FUNCTION_BLOCK FB_Camera EXTENDS FB_GCodeTool
VAR_INPUT
END_VAR
VAR_OUTPUT
END_VAR
VAR
	//SpecProperties
	rWorkingDistance		: REAL;
	bInvertWorkingDistance 	: BOOL;
	eLightOutput 			: E_TriggerOutput;
	nLightOutputChannel		: USINT;
	
	bCameraLightOn			: BOOL;
	
	bTakePicture			: BOOL;
	nStateA_TakePicture		: USINT;
	tDelayTakePicture		: TIME;
	timerTakePicture		: TON;
	nRequestArg1			: DINT;
	nRequestArg2			: DINT;
	nRequestArg3			: DINT;
	nRequestArg4			: DINT;	
END_VAR

IF bCameraLightOn THEN
	IF eLightOutput = E_TriggerOutput.MultiZOutput THEN
		fbMultiZDigiOut.M_On(nLightOutputChannel);
	ELSIF eLightOutput = E_TriggerOutput.MultiZPWM THEN
		fbMultiZPWM.M_On(nLightOutputChannel, 1000);
	END_IF
END_IF

IF eCurrentState = E_MachineState.MACHINESTATE_Active THEN
	IF bTakePicture THEN
		A_TakePicture();
		IF nStateA_TakePicture = 80 THEN
			nStateA_TakePicture := 0;
			bTakePicture := FALSE;
			M_RemoveListEntry(nSearchValue:= E_Action.ACTION_TakePicture);
		END_IF
	END_IF	
END_IF

SUPER^();

stProcessData.n32Data[7] := BOOL_TO_DINT(bCameraLightOn);
aObjProcData[nNotifyId] := stProcessData;

ACTION A_Reset:
nStateA_ResetSpec := 80;
SUPER^.A_Reset();
END_ACTION

ACTION A_Stop:
IF nStateA_Stop = 0 THEN
	IF bTakePicture AND nStateA_TakePicture < 70 THEN
		nStateA_TakePicture := 70;
	END_IF
	nStateA_Stop := 1;
END_IF

SUPER^.A_Stop();
END_ACTION

ACTION A_TakePicture:
IF nStateA_TakePicture = 0 THEN //Timer starten
	timerTakePicture(IN:= TRUE, PT:= tDelayTakePicture);
	IF timerTakePicture.Q THEN
		timerTakePicture(IN:= FALSE);
		stInterResponse.eInteractMessageType := E_InteractMessageType.INTERACTMES_NONE;
		stInteractRequest.eInteractMessageType := E_InteractMessageType.INTERACTMES_WaitForUser;
		stInteractRequest.nObjectId := nObjectID;
		stInteractRequest.nArg1 := nRequestArg1;
		stInteractRequest.nArg2 := nRequestArg2;
		stInteractRequest.nArg3 := nRequestArg3;
		stInteractRequest.nArg4 := nRequestArg4;
		nStateA_TakePicture := 1;
	END_IF
ELSIF nStateA_TakePicture = 1 THEN //Auf InteractResponse warten
	IF stInterResponse.eInteractMessageType = E_InteractMessageType.INTERACTMES_Continue OR 
							stInterResponse.eInteractMessageType = E_InteractMessageType.INTERACTMES_Cancel THEN
		stInteractRequest.eInteractMessageType := E_InteractMessageType.INTERACTMES_NONE;
		nStateA_TakePicture := 80;
	END_IF
ELSIF nStateA_TakePicture = 70 THEN //Abbrechen
	timerTakePicture(IN:= FALSE);
	stInteractRequest.eInteractMessageType := E_InteractMessageType.INTERACTMES_NONE;
	nStateA_TakePicture := 80;
END_IF
END_ACTION

METHOD FB_init : BOOL
VAR_INPUT
	bInitRetains : BOOL; // if TRUE, the retain variables are initialized (warm start / cold start)
	bInCopyCode : BOOL;  // if TRUE, the instance afterwards gets moved into the copy code (online change)
END_VAR
eObjectType := E_ObjectType.OBJECTTYPE_Camera;
eObjectGroup := E_ObjectGroup.OBJECTGROUP_MzTool OR E_ObjectGroup.OBJECTGROUP_Device;
END_METHOD

METHOD M_AddChild : ERRORID
VAR_INPUT
	pObject : POINTER TO FB_Object;
	nSlotNr	: UINT;	
	nIndex : INT;
END_VAR
//Kann folgende Objekte aufnehmen:
//Camera, Exposure
IF pObject > 0 THEN
	IF pObject^.P_eObjectType = E_ObjectType.OBJECTTYPE_Camera OR
		pObject^.P_eObjectType = E_ObjectType.OBJECTTYPE_DummyTool OR
		pObject^.P_eObjectType = E_ObjectType.OBJECTTYPE_Exposure THEN
		M_AddChild := SUPER^.M_AddChild(pObject,nSlotNr,nIndex);
	ELSE
		M_AddChild := E_ErrorIdObjMgmt.ERRORID_InvalidParentObject;
	END_IF
ELSE
	M_AddChild := E_ErrorIdObjMgmt.ERRORID_InvalidParentObject;
END_IF
END_METHOD

METHOD M_CancelAction
VAR_INPUT
	eAction : E_Action;
END_VAR
IF eAction = E_Action.ACTION_TakePicture THEN
	IF bTakePicture AND nStateA_TakePicture < 70 THEN
		nStateA_TakePicture := 70;
	END_IF
ELSE
	SUPER^.M_CancelAction(eAction);
END_IF
END_METHOD

METHOD M_CheckAction : ERRORID
VAR_INPUT
	refActionData 	: REFERENCE TO ST_ActionData;
	pCorrelObject	: POINTER TO FB_Object;
END_VAR

VAR
	pTarget : POINTER TO FB_TargetBase;
	pRack	: POINTER TO FB_Rack;
	pSlot	: POINTER TO FB_PieceSlot;
END_VAR
IF refActionData.eAction = E_Action.ACTION_TakePicture THEN
	RETURN;
ELSE
	M_CheckAction := SUPER^.M_CheckAction(refActionData, pCorrelObject);
END_IF
END_METHOD

METHOD M_ExeAction : ERRORID
VAR_INPUT
	refActionData : REFERENCE TO ST_ActionData;	
END_VAR
IF NOT (eCurrentState = E_MachineState.MACHINESTATE_Idle OR
	eCurrentState = E_MachineState.MACHINESTATE_Active OR
	eCurrentState = E_MachineState.MACHINESTATE_Ready) THEN
	M_ExeAction := E_ErrorIdCmd.ERRORID_InvalidState;
	RETURN;
END_IF

IF refActionData.eAction = E_Action.ACTION_SwitchLight THEN
	bCameraLightOn := DINT_TO_BOOL(refActionData.aParams[1]);
ELSIF refActionData.eAction = E_Action.ACTION_TakePicture THEN
	IF NOT bTakePicture THEN
		tDelayTakePicture := DINT_TO_TIME(refActionData.aParams[1]);
		nRequestArg1 := refActionData.aParams[2];
		nRequestArg2 := refActionData.aParams[3];
		nRequestArg3 := refActionData.aParams[4];
		nRequestArg4 := refActionData.aParams[5];
		
		fbList.A_AddHeadValue(hList := hList, putValue := E_Action.ACTION_TakePicture);
		bTakePicture := TRUE;
	END_IF
ELSE
	M_ExeAction := SUPER^.M_ExeAction(refActionData);
	RETURN;	
END_IF

bBusy := TRUE;
eCurrentState := E_MachineState.MACHINESTATE_Active;
END_METHOD

METHOD M_GetAllProps : ERRORID
VAR_INPUT
	refCmdData : REFERENCE TO  ST_CmdData;
END_VAR
SUPER^.M_GetAllProps(refCmdData);
nCurrentPropIndex := nCurrentPropIndex + 1;
refCmdData.n32Data[nCurrentPropIndex] := REAL_TO_DINT(rWorkingDistance);
nCurrentPropIndex := nCurrentPropIndex + 1;
refCmdData.n32Data[nCurrentPropIndex] := BOOL_TO_DINT(bInvertWorkingDistance);
nCurrentPropIndex := nCurrentPropIndex + 1;
refCmdData.n32Data[nCurrentPropIndex] := eLightOutput;
nCurrentPropIndex := nCurrentPropIndex + 1;
refCmdData.n32Data[nCurrentPropIndex] := nLightOutputChannel;
END_METHOD

METHOD M_SetAllProps : ERRORID
VAR_INPUT
	refCmdData : REFERENCE TO  ST_CmdData;
END_VAR
M_SetAllProps := SUPER^.M_SetAllProps(refCmdData);

IF M_SetAllProps > 0 THEN
	RETURN;
END_IF

//WorkingDistance
nCurrentPropIndex := nCurrentPropIndex + 1;
nSpecPropIndex := nCurrentPropIndex;
rWorkingDistance := DINT_TO_REAL(refCmdData.n32Data[nCurrentPropIndex]);
nCurrentPropIndex := nCurrentPropIndex + 1;
bInvertWorkingDistance := DINT_TO_BOOL(refCmdData.n32Data[nCurrentPropIndex]);

//LightOutput
nCurrentPropIndex := nCurrentPropIndex + 1;
eLightOutput := DINT_TO_USINT(refCmdData.n32Data[nCurrentPropIndex]);

//LightOutputChannel
nCurrentPropIndex := nCurrentPropIndex + 1;
nLightOutputChannel := DINT_TO_USINT(refCmdData.n32Data[nCurrentPropIndex]);

nNoOfProps := nCurrentPropIndex + 1;
END_METHOD

METHOD M_SetSingleProp : ERRORID
VAR_INPUT
	refCmdData : REFERENCE TO  ST_CmdData;
END_VAR
IF nSpecPropIndex = refCmdData.aHeader[1] THEN
	rWorkingDistance := DINT_TO_REAL(refCmdData.n32Data[0]);
ELSIF nSpecPropIndex + 1 = refCmdData.aHeader[1] THEN
	bInvertWorkingDistance := DINT_TO_BOOL(refCmdData.n32Data[0]);
ELSIF nSpecPropIndex + 3 = refCmdData.aHeader[1] THEN
	nLightOutputChannel := DINT_TO_USINT(refCmdData.n32Data[0]);
ELSE
	M_SetSingleProp := SUPER^.M_SetSingleProp(refCmdData);
END_IF
END_METHOD

PROPERTY P_stAbsPosTotal : ST_3DPoint
GET
VAR
	stPosTemp : ST_3DPoint;
END_VAR
stPosTemp := SUPER^.P_stAbsPosPhys;
IF bInvertWorkingDistance THEN
	stPosTemp.Z := stPosTemp.Z + rWorkingDistance;
ELSE
	stPosTemp.Z := stPosTemp.Z - rWorkingDistance;
END_IF
P_stAbsPosTotal := stPosTemp;
END_GET
END_PROPERTY

PROPERTY P_stCurrentPosTotal : ST_3DPoint
GET
VAR
	stPosTemp : ST_3DPoint;
END_VAR
stPosTemp := P_stCurrentPosPhys;
IF bInvertWorkingDistance THEN
	stPosTemp.Z := stPosTemp.Z + rWorkingDistance;
ELSE
	stPosTemp.Z := stPosTemp.Z - rWorkingDistance;
END_IF
P_stCurrentPosTotal := stPosTemp;
END_GET
END_PROPERTY

END_FUNCTION_BLOCK

(* stored: Version 1.1.0.1, ProductVersion 3.1.4024.11
   POU FB_Camera: Id {6d1727e9-21d6-47ab-aac6-925ca4a23f77}, SpecialFunc None
   Action A_Reset: Id {43cf20d4-7297-4beb-a482-862479609b93}
   Action A_Stop: Id {44fa0f71-374f-45e3-97ba-21c728d998ed}
   Action A_TakePicture: Id {c447fb64-ca66-4994-a719-68951c0efcd5}
   Method FB_init: Id {87c6810b-20b1-4848-9659-f4d11b203ab8}
   Method M_AddChild: Id {7fbea080-b919-479e-82a2-845d1d7d009a}
   Method M_CancelAction: Id {913818c3-739d-47c2-8f9f-61bcaba57241}
   Method M_CheckAction: Id {9fbc6bc5-2680-450f-a2c1-5f570e5cb51f}
   Method M_ExeAction: Id {ff212081-912a-4cff-b8c5-f2d1a4eaf519}
   Method M_GetAllProps: Id {ee3bbb9b-aa27-457d-998b-0872851fe694}
   Method M_SetAllProps: Id {5942dde0-2cc4-4175-8189-ee55fd5bd1a7}
   Method M_SetSingleProp: Id {5a3b6e7d-63ee-40a8-b359-252b2712110d}
   Property P_stAbsPosTotal: Id {05053f60-fb68-41b0-bdd5-cdb432e72623}
   Get Get: Id {9c92bc8d-37ca-4da7-8b85-6ccb9cf23d05}
   Property P_stCurrentPosTotal: Id {ead232df-6902-4ba7-b56f-60f77812030d}
   Get Get: Id {af8adb17-0a1d-4c90-8336-a1cf5f4690b9} *)
